FUNCTION_BLOCK FB_SimulatedIn_DG IMPLEMENTS ITF_Regelschuif_IN_DG

VAR
	internalState : sint;
END_VAR

{warning 'Add method implementation '}
METHOD get : SINT
get := internalState;
END_METHOD

END_FUNCTION_BLOCK

(* stored: Version 1.1.0.1, ProductVersion 3.1.4026.8
   POU FB_SimulatedIn_DG: Id {63c47254-f5df-4fce-ac77-dfc31f6df536}, SpecialFunc None
   Method get: Id {6aed3395-d16f-4f02-8d40-c7ce69b68c06} *)
